# EPICS StreamDevice protocol: db/afg3000.proto
# This is a protocol file for AFG3000 series
#
terminator = LF;
intFuncFormat = "%{SIN|SQU|TRI|RAMP|NRAM|PRN|USER|USER2|USER3|USER4|EMEM|EFIL}";
srcFuncFormat = "%#{SQU=1|PULS|RAMP|PRN|DC|SINC|GAUS|LOR|ERIS|EDEC|HAV|USER2=13|USER3|USER4|EMEM|EFIL|SIN=0|USER=12}";

# Output commands
# @param $1 channel number

getOutputImpedance {
    out "OUTP\$1:IMP?";
        in  "%f";
	}
	setOutputImpedance {
	    out "OUTP\$1:IMP %f";
	        @init{getOutputImpedance;};
		}

getOutputPolarity {
    out "OUTP\$1:POL?";
        in  "%{NORM|INV}";
	}
	setOutputPolarity {
	    out "OUTP\$1:POL %{NORM|INV}";
	        @init{getOutputPolarity;};
		}

getOutputState {
    out "OUTP\$1:STAT?";
        in  "%d";
	}
	setOutputState {
	    out "OUTP\$1:STAT %{OFF|ON}";
	        @init{getOutputState;};
		}

getOutputTriggerMode {
    out "OUTP:TRIG:MODE?";
        in  "%{TRIG|SYNC}";
	}
	setOutputTriggerMode {
	    out "OUTP:TRIG:MODE %{TRIG|SYNC}";
	        @init{getOutputTriggerMode;};
		}

# Source commands

## Reference Oscillator source
getSourceROSource {
    out "SOUR:ROSC:SOUR?";
        in  "%{INT|EXT}";
	}
	setSourceROSource {
	    out "SOUR:ROSC:SOUR %{INT|EXT}";
	        @init{getSourceROSource;};
		}

## Amplitude modulation
getSourceAMState {
    out "SOUR\$1:AM:STAT?";
        in  "%d";
	}
	setSourceAMState {
	    out "SOUR\$1:AM:STAT %{OFF|ON}";
	        @init{getSourceAMState;};
		}

getSourceFrequency {
    out "SOUR\$1:FREQ:FIX?";
        in  "%f";
	}
	setSourceFrequency {
	    out "SOUR\$1:FREQ:FIX %f";
	        @init{getSourceFrequency;};
		}

getSourceAMInternalFrequency {
    out "SOUR\$1:AM:INT:FREQ?";
        in  "%f";
	}
	setSourceAMInternalFrequency {
	    out "SOUR\$1:AM:INT:FREQ %f";
	        @init{getSourceAMInternalFrequency;};
		}

getSourceAMInternalFunction {
    out "SOUR\$1:AM:INT:FUNC?";
        in  $intFuncFormat;
	}
	setSourceAMInternalFunction {
	    out "SOUR\$1:AM:INT:FUNC " $intFuncFormat;
	        @init{getSourceAMInternalFunction;};
		}

getSourceAMInternalFunctionEFile {
    out "SOUR\$1:AM:INT:FUNC:EFIL?";
        in  "\"%[^\"]\"";
	}
	setSourceAMInternalFunctionEFile {
	    out "SOUR\$1:AM:INT:FUNC:EFIL \"%s\"";
	        @init{getSourceAMInternalFunctionEFile;};
		}

getSourceAMSource {
    out "SOUR\$1:AM:SOUR?";
        in  "%{INT|EXT}";
	}
	setSourceAMSource {
	    out "SOUR\$1:AM:SOUR %{INT|EXT}";
	        @init{getSourceAMSource;};
		}

getSourceAMDepth {
    out "SOUR\$1:AM:DEPT?";
        in  "%f";
	}
	setSourceAMDepth {
	    out "SOUR\$1:AM:DEPT %f";
	        @init{getSourceAMDepth;};
		}

## Burst mode
getSourceBurstMode {
    out "SOUR\$1:BURS:MODE?";
        in  "%{TRIG|GAT}";
	}
	setSourceBurstMode {
	    out "SOUR\$1:BURS:MODE %{TRIG|GAT}";
	        @init{getSourceBurstMode;};
		}

getSourceBurstNCycles {
    out "SOUR\$1:BURS:NCYC?";
        in  "%f";
	}
	setSourceBurstNCycles {
	    out "SOUR\$1:BURS:NCYC %f";
	        @init{getSourceBurstNCycles;};
		}

getSourceBurstTdelay {
    out "SOUR\$1:BURS:TDEL?";
        in  "%g";
	}
	setSourceBurstTdelay {
	    out "SOUR\$1:BURS:TDEL %g";
	        @init{getSourceBurstTdelay;};
		}

getSourceBurstState {
    out "SOUR\$1:BURS:STAT?";
        in  "%d";
	}
	setSourceBurstState {
	    out "SOUR\$1:BURS:STAT %{OFF|ON}";
	        @init{getSourceBurstState;};
		}

## Combined feed
# Different options on the two channels.
# AFG3051C only has one channel, records to channel 2 are not done.
getSourceCombineFeed1 {
    out "SOUR1:COMB:FEED?";
        in  "\"%{NOIS|EXT|BOTH|}\"";
	}
	setSourceCombineFeed1 {
	    out "SOUR1:COMB:FEED \"%{NOIS|EXT|BOTH|}\"";
	        @init{getSourceCombineFeed1;};
		}

getSourceCombineFeed2 {
    out "SOUR2:COMB:FEED?";
        in  "%{\"NOIS\"|\"\"}";
	}
	setSourceCombineFeed2 {
	    out "SOUR2:COMB:FEED %{\"NOIS\"|\"\"}";
	        @init{getSourceCombineFeed2;};
		}

## Frequency modulation
getSourceFMInternalFrequency {
    out "SOUR\$1:FM:INT:FREQ?";
        in  "%f";
	}
	setSourceFMInternalFrequency {
	    out "SOUR\$1:FM:INT:FREQ %f";
	        @init{getSourceFMInternalFrequency;};
		}

getSourceFMInternalFunction {
    out "SOUR\$1:FM:INT:FUNC?";
        in  $intFuncFormat;
	}
	setSourceFMInternalFunction {
	    out "SOUR\$1:FM:INT:FUNC " $intFuncFormat;
	        @init{getSourceFMInternalFunction;};
		}

getSourceFMInternalFunctionEfile {
    out "SOUR\$1:FM:INT:FUNC:EFIL?";
        in  "\"%[^\"]\"";
	}
	setSourceFMInternalFunctionEfile {
	    out "SOUR\$1:FM:INT:FUNC:EFIL \"%s\"";
	        @init{getSourceFMInternalFunctionEfile;};
		}

getSourceFMSource {
    out "SOUR\$1:FM:SOUR?";
        in  "%{INT|EXT}";
	}
	setSourceFMSource {
	    out "SOUR\$1:FM:SOUR %{INT|EXT}";
	        @init{getSourceFMSource;};
		}

getSourceFMState {
    out "SOUR\$1:FM:STAT?";
        in  "%d";
	}
	setSourceFMState {
	    out "SOUR\$1:FM:STAT %{OFF|ON}";
	        @init{getSourceFMState;};
		}

getSourceFMDeviation {
    out "SOUR\$1:FM:DEV?";
        in  "%f";
	}
	setSourceFMDeviation {
	    out "SOUR\$1:FM:DEV %f";
	        @init{getSourceFMDeviation;};
		}

getSourceFrequencyCenter {
    out "SOUR\$1:FREQ:CENT?";
        in  "%f";
	}
	setSourceFrequencyCenter {
	    out "SOUR\$1:FREQ:CENT %f";
	        @init{getSourceFrequencyCenter;};
		}

getSourceFrequencyConcurrent{
    out "SOUR\$1:FREQ:CONC:STAT?";
        in  "%d";
	}
	setSourceFrequencyConcurrent {
	    out "SOUR\$1:FREQ:CONC:STAT %{OFF|ON}";
	        @init{getSourceFrequencyConcurrent;};
		}

getSourceFrequencyMode {
    out "SOUR\$1:FREQ:MODE?";
        in  "%{CW|SWE}";
	}
	setSourceFrequencyMode {
	    out "SOUR\$1:FREQ:MODE %{CW|SWE}";
	        @init{getSourceFrequencyMode;};
		}

getSourceFrequencySpan {
    out "SOUR\$1:FREQ:SPAN?";
        in  "%g";
	}
	setSourceFrequencySpan {
	    out "SOUR\$1:FREQ:SPAN %g";
	        @init{getSourceFrequencySpan;};
		}

getSourceFrequencyStart {
    out "SOUR\$1:FREQ:STAR?";
        in  "%g";
	}
	setSourceFrequencyStart {
	    out "SOUR\$1:FREQ:STAR %g";
	        @init{getSourceFrequencyStart;};
		}

getSourceFrequencyStop {
    out "SOUR\$1:FREQ:STOP?";
        in  "%g";
	}
	setSourceFrequencyStop {
	    out "SOUR\$1:FREQ:STOP %g";
	        @init{getSourceFrequencyStop;};
		}

getSourceFrequencyFixed{
    out "SOUR\$1:FREQ:FIX?";
        in  "%g";
	}
	setSourceFrequencyFixed{
	    out "SOUR\$1:FREQ:FIX %g";
	        @init{getSourceFrequencyFixed;};
		}

getSourceFSKeyInternalRate {
    out "SOUR\$1:FSK:INT:RATE?";
        in  "%g";
	}
	setSourceFSKeyInternalRate {
	    out "SOUR\$1:FSK:INT:RATE %g";
	        @init{getSourceFSKeyInternalRate;};
		}

getSourceFSKeySource {
    out "SOUR\$1:FSK:SOUR?";
        in  "%{INT|EXT}";
	}
	setSourceFSKeySource {
	    out "SOUR\$1:FSK:SOUR %{INT|EXT}";
	        @init{getSourceFSKeySource;};
		}

getSourceFSKeyState{
    out "SOUR\$1:FSK:STAT?";
        in  "%d";
	}
	setSourceFSKeyState {
	    out "SOUR\$1:FSK:STAT %{OFF|ON}";
	        @init{getSourceFSKeyState;};
		}

getSourceFSKeyFrequency {
    out "SOUR\$1:FSK:FREQ?";
        in  "%g";
	}
	setSourceFSKeyFrequency {
	    out "SOUR\$1:FSK:FREQ %g";
	        @init{getSourceFSKeyFrequency;};
		}

getSourceFunctionRampSymmetry {
    out "SOUR\$1:FUNC:RAMP:SYMM?";
        in  "%f";
	}
	setSourceFunctionRampSymmetry {
	    out "SOUR\$1:FUNC:RAMP:SYMM %f";
	        @init{getSourceFunctionRampSymmetry;};
		}

getSourceFunctionShape {
    out "SOUR\$1:FUNC:SHAP?";
        in  $srcFuncFormat;
	}
	setSourceFunctionShape {
	    out "SOUR\$1:FUNC:SHAP " $srcFuncFormat;
	        @init{getSourceFunctionShape;};
		}

getSourceFunctionEFile {
    out "SOUR\$1:FUNC:EFIL?";
        in  "\"%[^\"]\"";
	}
	setSourceFunctionEFile {
	    out "SOUR\$1:FUNC:EFIL \"%s\"";
	        @init{getSourceFunctionEFile;};
		}

sourcePhaseInitiate {
    out "SOUR\$1:PHAS:INIT";
    }

getSourcePhaseAdjust {
    out "SOUR\$1:PHAS:ADJ?";
        in  "%g";
	}
	setSourcePhaseAdjust {
	    out "SOUR\$1:PHAS:ADJ %g";
	        @init{getSourcePhaseAdjust;};
		}

getSourcePMInternalFrequency{
    out "SOUR\$1:PM:INT:FREQ?";
        in  "%g";
	}
	setSourcePMInternalFrequency {
	    out "SOUR\$1:PM:INT:FREQ %g";
	        @init{getSourcePMInternalFrequency;};
		}

getSourcePMInternalFunction{
    out "SOUR\$1:PM:INT:FUNC?";
        in $intFuncFormat;
	}
	setSourcePMInternalFunction {
	    out "SOUR\$1:PM:INT:FUNC " $intFuncFormat;
	        @init{getSourcePMInternalFunction;};
		}

getSourcePMInternalFunctionEfile{
    out "SOUR\$1:PM:INT:FUNC:EFIL?";
        in  "\"%[^\"]\"";
	}
	setSourcePMInternalFunctionEfile{
	    out "SOUR\$1:PM:INT:FUNC:EFIL \"%s\"";
	        @init{getSourcePMInternalFunctionEfile;};
		}

getSourcePMSource {
    out "SOUR\$1:PM:SOUR?";
        in  "%{INT|EXT}";
	}
	setSourcePMSource {
	    out "SOUR\$1:PM:SOUR %{INT|EXT}";
	        @init{getSourcePMSource;};
		}

getSourcePMState {
    out "SOUR\$1:PM:STAT?";
        in  "%d";
	}
	setSourcePMState {
	    out "SOUR\$1:PM:STAT %{OFF|ON}";
	        @init{getSourcePMState;};
		}

getSourcePMDeviation{
    out "SOUR\$1:PM:DEV?";
        in  "%g";
	}
	setSourcePMDeviation {
	    out "SOUR\$1:PM:DEV %g";
	        @init{getSourcePMDeviation;};
		}

# Only channel 3 and 4.
getSourcePower {
    out "SOUR\$1:POW?";
        in "%f";
	}
	setSourcePower {
	    out "SOUR\$1:POW %f";
	        @init{getSourcePower;};
		}

getSourcePulseDCycle {
    out "SOUR\$1:PULS:DCYC?";
        in  "%f";
	}
	setSourcePulseDCycle {
	    out "SOUR\$1:PULS:DCYC %f";
	        @init{getSourcePulseDCycle;};
		}

getSourcePulseDelay {
    out "SOUR\$1:PULS:DEL?";
        in  "%g";
	}
	setSourcePulseDelay {
	    out "SOUR\$1:PULS:DEL %g";
	        @init{getSourcePulseDelay;};
		}

getSourcePulseHold {
    out "SOUR\$1:PULS:HOLD?";
        in  "%{WIDT|DUTY}";
	}
	setSourcePulseHold {
	    out "SOUR\$1:PULS:HOLD %{WIDT|DUTY}";
	        @init{getSourcePulseHold;};
		}

getSourcePulsePeriod {
    out "SOUR\$1:PULS:PER?";
        in  "%g";
	}
	setSourcePulsePeriod {
	    out "SOUR\$1:PULS:PER %g";
	        @init{getSourcePulsePeriod;};
		}

getSourcePulseTransitionLeading {
    out "SOUR\$1:PULS:TRAN:LEAD?";
        in  "%g";
	}
	setSourcePulseTransitionLeading {
	    out "SOUR\$1:PULS:TRAN:LEAD %g";
	        @init{getSourcePulseTransitionLeading;};
		}

getSourcePulseTransitionTrailing {
    out "SOUR\$1:PULS:TRAN:TRA?";
        in  "%g";
	}
	setSourcePulseTransitionTrailing {
	    out "SOUR\$1:PULS:TRAN:TRA %g";
	        @init{getSourcePulseTransitionTrailing;};
		}

getSourcePulseWidth {
    out "SOUR\$1:PULS:WIDT?";
        in  "%g";
	}
	setSourcePulseWidth {
	    out "SOUR\$1:PULS:WIDT %g";
	        @init{getSourcePulseWidth;};
		}

getSourcePWMInternalFrequency {
    out "SOUR\$1:PWM:INT:FREQ?";
        in  "%g";
	}
	setSourcePWMInternalFrequency {
	    out "SOUR\$1:PWM:INT:FREQ %g";
	        @init{getSourcePWMInternalFrequency;};
		}

getSourcePWMInternalFunction {
    out "SOUR\$1:PWM:INT:FUNC?";
        in $intFuncFormat;
	}
	setSourcePWMInternalFunction {
	    out "SOUR\$1:PWM:INT:FUNC " $intFuncFormat;
	        @init{getSourcePWMInternalFunction;};
		}

getSourcePWMInternalFunctionEfile {
    out "SOUR\$1:PWM:INT:FUNC:EFIL?";
        in  "\"%[^\"]\"";
	}
	setSourcePWMInternalFunctionEfile {
	    out "SOUR\$1:PWM:INT:FUNC:EFIL \"%s\"";
	        @init{getSourcePWMInternalFunctionEfile;};
		}

getSourcePWMSource {
    out "SOUR\$1:PWM:SOUR?";
        in  "%{INT|EXT}";
	}
	setSourcePWMSource {
	    out "SOUR\$1:PWM:SOUR %{INT|EXT}";
	        @init{getSourcePWMSource;};
		}

getSourcePWMState {
    out "SOUR\$1:PWM:STAT?";
        in  "%d";
	}
	setSourcePWMState {
	    out "SOUR\$1:PWM:STAT %{OFF|ON}";
	        @init{getSourcePWMState;};
		}

getSourcePWMDeviationDCycle {
    out "SOUR\$1:PWM:DEV:DCYC?";
        in  "%f";
	}
	setSourcePWMDeviationDCycle {
	    out "SOUR\$1:PWM:DEV:DCYC %f";
	        @init{getSourcePWMDeviationDCycle;};
		}

getSourceSweepHTime {
    out "SOUR\$1:SWE:HTIM?";
        in  "%g";
	}
	setSourceSweepHTime {
	    out "SOUR\$1:SWE:HTIM %g";
	        @init{getSourceSweepHTime;};
		}

getSourceSweepMode {
    out "SOUR\$1:SWE:MODE?";
        in  "%{AUTO|MAN}";
	}
	setSourceSweepMode {
	    out "SOUR\$1:SWE:MODE %{AUTO|MAN}";
	        @init{getSourceSweepMode;};
		}

getSourceSweepRTime {
    out "SOUR\$1:SWE:RTIM?";
        in  "%g";
	}
	setSourceSweepRTime {
	    out "SOUR\$1:SWE:RTIM %g";
	        @init{getSourceSweepRTime;};
		}

getSourceSweepSpacing {
    out "SOUR\$1:SWE:SPAC?";
        in  "%{LIN|LOG}";
	}
	setSourceSweepSpacing {
	    out "SOUR\$1:SWE:SPAC %{LIN|LOG}";
	        @init{getSourceSweepSpacing;};
		}

getSourceSweepTime {
    out "SOUR\$1:SWE:TIME?";
        in  "%g";
	}
	setSourceSweepTime {
	    out "SOUR\$1:SWE:TIME %g";
	        @init{getSourceSweepTime;};
		}

getSourceVoltageConcurrentState {
    out "SOUR\$1:VOLT:CONC:STAT?";
        in  "%d";
	}
	setSourceVoltageConcurrentState {
	    out "SOUR\$1:VOLT:CONC:STAT %{OFF|ON}";
	        @init{getSourceVoltageConcurrentState;};
		}

getSourceVoltageLimitHigh {
    out "SOUR\$1:VOLT:LIM:HIGH?";
        in  "%g";
	}
	setSourceVoltageLimitHigh {
	    out "SOUR\$1:VOLT:LIM:HIGH %g";
	        @init{getSourceVoltageLimitHigh;};
		}

getSourceVoltageLimitLow {
    out "SOUR\$1:VOLT:LIM:LOW?";
        in  "%g";
	}
	setSourceVoltageLimitLow {
	    out "SOUR\$1:VOLT:LIM:LOW %g";
	        @init{getSourceVoltageLimitLow;};
		}

getSourceVoltageUnit {
    out "SOUR\$1:VOLT:UNIT?";
        in  "%{VPP|VRMS|DBM}";
	}
	setSourceVoltageUnit {
	    out "SOUR\$1:VOLT:UNIT %{VPP|VRMS|DBM}";
	        @init{getSourceVoltageUnit;};
		}

getSourceVoltageHigh {
    out "SOUR\$1:VOLT:HIGH?";
        in  "%g";
	}
	setSourceVoltageHigh {
	    out "SOUR\$1:VOLT:HIGH %g";
	        @init{getSourceVoltageHigh;};
		}

getSourceVoltageLow {
    out "SOUR\$1:VOLT:LOW?";
        in  "%g";
	}
	setSourceVoltageLow {
	    out "SOUR\$1:VOLT:LOW %g";
	        @init{getSourceVoltageLow;};
		}

getSourceVoltageOffset {
    out "SOUR\$1:VOLT:OFFS?";
        in  "%g";
	}
	setSourceVoltageOffset {
	    out "SOUR\$1:VOLT:OFFS %g";
	        @init{getSourceVoltageOffset;};
		}

getSourceVoltageAmplitude {
    out "SOUR\$1:VOLT?";
        in  "%g";
	}
	setSourceVoltageAmplitude {
	    out "SOUR\$1:VOLT %g";
	        @init{getSourceVoltageAmplitude;};
		}

# System commands
getIdentification {
    out "*IDN?";
        in  "%[^,],%(\$1-IMDL)[^,],%(\$1-ISN)[^,],%(\$1-IFW)[^,]";
	}

reset {
    out "*RST";
    }

# Data commands
getDataCatalog {
    Separator=",";
        out "DATA:CAT?";
	    in  "\"%[^\"]\"";
	    }

# Copy content from source to target memories.
# $1 Target  (EMEM|USER|USER2|USER3|USER4)
# $2 Source  (EMEM|USER|USER2|USER3|USER4)
setDataCopy {
    out "DATA:COPY \$1,\$2";
    }

# $1 Field which contains the number of digits in NORD.
getDataData {
    out "DATA:DATA? EMEM";
        in  "%s";
	}
	setDataData {
	    out "TRACE:DATA EMEM, #42000\$1";
	    }

setDataDelete{}
getDataDelete{}

setDataDefine{}
getDataDefine{}

setDataLock{}
getDataLock{}

setDataPoints{}
getDataPoints{}

setDataDataLine{}
getDataDataLine{}

setDataDataValue{}
getDataDataValue{}

# Trigger commands
getTriggerSlope {
    out "TRIG:SLOP?";
        in  "%{POS|NEG}";
	}
	setTriggerSlope {
	    out "TRIG:SLOP %{POS|NEG}";
	        @init{getTriggerSlope;};
		}

getTriggerSource {
    out "TRIG:SOUR?";
        in  "%{TIM|EXT}";
	}
	setTriggerSource {
	    out "TRIG:SOUR %{TIM|EXT}";
	        @init{getTriggerSource;};
		}

getTriggerTimer {
    out "TRIG:TIM?";
        in  "%g";
	}
	setTriggerTimer {
	    out "TRIG:TIM %g";
	        @init{getTriggerTimer;};
		}

trigger {
    out "TRIG";
    }
